FUNCTION_BLOCK PUBLIC FB_PizzaAmericanStyle IMPLEMENTS I_Pizza
VAR_INPUT
END_VAR
VAR_OUTPUT
END_VAR
VAR
END_VAR

METHOD PUBLIC GetPrice : LREAL
VAR_INPUT
END_VAR
GetPrice := 4.2;
END_METHOD

END_FUNCTION_BLOCK

(* stored: Version 1.1.0.1, ProductVersion 3.1.4022.12
   POU FB_PizzaAmericanStyle: Id {cb40c609-3f26-4c2a-bce6-73adf6f1a66e}, SpecialFunc None
   Method GetPrice: Id {b18f3b20-fa10-4361-988b-e78b81243b43} *)
